{attribute 'qualified_only'}
{attribute 'strict'}
TYPE PtWeekDay :
(
	MONDAY := 0,
    TUESDAY := 1,
    WEDNESDAY := 2,
    THURSDAY := 3,
    FRIDAY := 4,
    SATURDAY := 5,
    SUNDAY := 6
);
END_TYPE

(* stored: Version 1.1.0.1, ProductVersion 3.1.4024.12
   EnumerationTextList PtWeekDay: Id {315bc762-1f22-4d0c-ae7a-afa497230d4a} *)
